FUNCTION_BLOCK FB_AnalogOutput
VAR_INPUT
END_VAR
VAR_INPUT
	fValue		: REAL; //input value	
END_VAR
VAR_OUTPUT
	nValue 		: INT; //converted value
END_VAR
VAR
	fUpperLimit : REAL; //upper limit of value range
	fLowerLimit : REAL; //lower limit of value range
END_VAR

// conversion from Bit value to actual value
nValue := REAL_TO_INT((fValue-fLowerLimit)/(fUpperLimit-fLowerLimit)*32767);

METHOD FB_init : BOOL
VAR_INPUT
	bInitRetains : BOOL; // if TRUE, the retain variables are initialized (warm start / cold start)
	bInCopyCode : BOOL;  // if TRUE, the instance afterwards gets moved into the copy code (online change)
	fUpperLimit : REAL; //upper limit of value range
	fLowerLimit : REAL; //lower limit of value range
END_VAR
//copy input values to internal variables
THIS^.fUpperLimit := fUpperLimit;
THIS^.fLowerLimit := fLowerLimit;
END_METHOD

END_FUNCTION_BLOCK

(* stored: Version 1.1.0.1, ProductVersion 3.1.4024.10
   POU FB_AnalogOutput: Id {e8cc816e-9340-40fa-8115-6e9fa806b2a4}, SpecialFunc None
   Method FB_init: Id {a1fc4530-5ecd-48d2-b2ae-0a43985b9150} *)
